(* CODESYS project Untitled2.project

Project tree, tasks and I/O mapping:
  Device : CODESYS Control Win V3, 3S - Smart Software Solutions GmbH, version 3.5.15.30
    application Application
      libraries: Standard, * (System)
      task MainTask (cyclic, interval t#20ms, priority 1) calls PLC_PRG
      program PLC_PRG [ST]
      function block MyFB [ST]
      program POU [FBD]
*)

// Device/Application/PLC_PRG
PROGRAM PLC_PRG
VAR
	A: REAL := 11;
	B: REAL := 5;
	Sum: REAL;
	Subtr: REAL;
	SumAndSubtract: MyFB;
END_VAR

SumAndSubtract(num1 := A, num2 := B);

Sum := SumAndSubtract.AddResult;
Subtr := SumAndSubtract.SubResult;

END_PROGRAM

// Device/Application/MyFB
FUNCTION_BLOCK MyFB
VAR_INPUT
	num1: REAL;
	num2: REAL;
END_VAR
VAR_OUTPUT
	AddResult: REAL;
	SubResult: REAL;
END_VAR
VAR
END_VAR

AddResult := num1 + num2;
SubResult := num1 - num2;

END_FUNCTION_BLOCK

// Device/Application/POU
PROGRAM POU
VAR
	SumAndSub: MyFB;
END_VAR

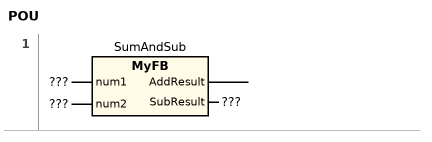
// NETWORK 1
SumAndSub(); // MyFB

END_PROGRAM
